TYPE TTableSide :
	(
		TS_A := 0,
		TS_B,
		TS_Moving
	);
END_TYPE

(* stored: Version 1.1.0.1, ProductVersion 3.1.4022.12
   DUT TTableSide: Id {fedbf240-0bdc-429f-93e6-2935e9380630} *)
